FUNCTION_BLOCK DefaultContext EXTENDS TcoCore.TcoContext
VAR
	_wpfCyclinder : TcoPneumatics.Cylinder(THIS^);
	_wpfCyclinder_1 : TcoPneumatics.Cylinder(THIS^);
	_wpfCyclinder_2 : TcoPneumatics.Cylinder(THIS^);
	_wpfCyclinder_3 : TcoPneumatics.Cylinder(THIS^);
END_VAR

METHOD PROTECTED  Main
_wpfCyclinder(inAtHomePos := IO.A1[0],
	inAtWorkPos := IO.A1[1],
	outToHomePos => IO.A2[0],
	outToWorkPos => IO.A2[1]);

_wpfCyclinder_1();
_wpfCyclinder_2();
_wpfCyclinder_3();
END_METHOD

END_FUNCTION_BLOCK

(* stored: Version 1.1.0.1, ProductVersion 3.1.4024.6
   POU DefaultContext: Id {9566aeb0-f006-4c52-ace4-7824786d839b}, SpecialFunc None
   Method Main: Id {f765357f-253d-4bf2-baf0-fad144fcb997} *)
